(* IEC 61131-3 sources: AXOpen/src/showcase/app/src/core/AXOpen.AxoSequencer, 2 files *)

(* ---- AxoSequencerDocuExample.st ---- *)
USING AXOpen.Core;

NAMESPACE AxoSequencerExamples
    {S7.extern=ReadWrite}
    CLASS AxoSequencerDocuExample EXTENDS  AXOpen.Core.AxoObject
        VAR PUBLIC
            _mySequencer : AXOpen.Core.AxoSequencer;
            _step_1 : AxoStep;
            _step_2 : AxoStep;
            _step_3 : AxoStep;
            _myCounter : ULINT;
        END_VAR

        //<Initialize>
        METHOD PUBLIC Initialize
            _mySequencer.Run(THIS);
        END_METHOD
        //</Initialize>

        METHOD PUBLIC Execute
            //<Open>
            THIS.Initialize();
            IF _mySequencer.Open() THEN
                //All sequence logic needs to be placed inside the condition
                _myCounter := _myCounter + ULINT#1;

                IF _step_1.Execute(_mySequencer) THEN
                    IF (_myCounter > ULINT#50) THEN
                        _mySequencer.MoveNext();
                    END_IF;
                END_IF;

                IF _step_2.Execute(_mySequencer) THEN
                    IF (_myCounter > ULINT#100) THEN
                        _mySequencer.MoveNext();
                    END_IF;
                END_IF;

                IF _step_3.Execute(_mySequencer) THEN
                    IF (_myCounter > ULINT#150) THEN
                        _myCounter := ULINT#0;
                        _mySequencer.CompleteSequence();
                    END_IF;
                END_IF;
            END_IF;
            //</Open>
        END_METHOD

        METHOD StepExamples
            //<SimpleStep>
            IF _step_1.Execute(_mySequencer) THEN
                _myCounter := _myCounter + ULINT#1;
                // do something
                IF (_myCounter MOD ULINT#5) = ULINT#0 THEN
                    // continue to the next step of the sequence
                    _mySequencer.MoveNext();
                END_IF;
            END_IF;
            //</SimpleStep>

            //<EnableStep>
                IF _step_2.Execute(coord := _mySequencer, Enable := _myCounter <= ULINT#20) THEN
                    _myCounter := _myCounter + ULINT#1;
                    IF _myCounter = ULINT#20 THEN
                        // Jumping to step 1. As it is jumping backwards, the execution of step 1
                        // is going to be started in the next context cycle.
                        _mySequencer.RequestStep(_step_1);
                    END_IF;
                END_IF;
            //</EnableStep>

            //<FullStep>
                IF _step_3.Execute(coord := _mySequencer, Enable := TRUE, Description := '<#Process data#>' ) THEN
                    _myCounter := _myCounter + ULINT#1;
                    IF (_myCounter MOD ULINT#7) = ULINT#0 THEN
                        // Finalize the sequence and initiate the execution from the first step.
                        _mySequencer.CompleteSequence();
                    END_IF;
                END_IF;
            //</FullStep>
        END_METHOD

        //<SequenceMode>
        METHOD SequenceModeExamples
            // RunOnce: sequence executes once and stays in Done state
            _mySequencer.SequenceMode := eAxoSequenceMode#RunOnce;

            // Cyclic: sequence restarts automatically after CompleteSequence
            _mySequencer.SequenceMode := eAxoSequenceMode#Cyclic;
        END_METHOD
        //</SequenceMode>
    END_CLASS
END_NAMESPACE

(* ---- AxoSequencerExample.st ---- *)
USING AXOpen.Core;

NAMESPACE AxoSequencerExamples

    {S7.extern=ReadWrite}
    CLASS SequencerExample EXTENDS  AXOpen.Core.AxoObject
        VAR PUBLIC
            {#ix-set:AttributeName = "<#Sequencer example#>"}
            coord : AxoSequencer;
            Counter : ULINT;
            {#ix-set:AttributeName = "<#MicroStep-should be set to zero when entering new step#>"}
            MicroStep : UINT;
        END_VAR

        VAR PUBLIC
            {#ix-set:Description = "Step number one"}
            step_1 : AxoStep;
            {#ix-set:Description = "Step number two"}
            step_2 : AxoStep;
            {#ix-set:Description = "Step number three"}
            step_3 : AxoStep;
            {#ix-set:Description = "Step number four"}
            step_4 : AxoStep;
            {#ix-set:Description = "Step number five"}
            step_5 : AxoStep;
            {#ix-set:Description = "Step number six"}
            step_6 : AxoStep;
            {#ix-set:Description = "Step number seven"}
            step_7 : AxoStep;
            {#ix-set:Description = "Step number eight"}
            step_8 : AxoStep;
            {#ix-set:Description = "Step number nine"}
            step_9 : AxoStep;
            {#ix-set:Description = "Step number ten"}
            step_10 : AxoStep;
            Enable : ARRAY[1..10] OF BOOL :=[10(TRUE)];
        END_VAR

        METHOD PUBLIC Execute
            coord.Run(THIS);

            IF coord.Open() THEN

                IF(step_1.Execute(coord,Enable[1], 'Step_1')) THEN
                    IF step_1.IsFirstEntryToStep() THEN
                        Counter := ULINT#100;
                    END_IF;
                    Counter := Counter + ULINT#1;
                    IF(Counter >= ULINT#200 ) THEN
                        Counter := ULINT#0;
                        coord.MoveNext();
                    END_IF;
                END_IF;

                IF(step_2.Execute(coord,Enable[2], 'Step_2')) THEN
                    IF step_2.IsFirstEntryToStep() THEN
                        Counter := ULINT#200;
                    END_IF;
                    Counter := Counter + ULINT#1;
                    IF(Counter >= ULINT#300 ) THEN
                        Counter := ULINT#0;
                        coord.MoveNext();
                    END_IF;
                END_IF;

                IF(step_3.Execute(coord,Enable[3], 'Step_3')) THEN
                    IF step_3.IsFirstEntryToStep() THEN
                        Counter := ULINT#300;
                    END_IF;
                    Counter := Counter + ULINT#1;
                    IF(Counter >= ULINT#400 ) THEN
                        Counter := ULINT#0;
                        coord.MoveNext();
                    END_IF;
                END_IF;

                IF(step_4.Execute(coord,Enable[4], 'Step_4')) THEN
                    IF step_4.IsFirstEntryToStep() THEN
                        Counter := ULINT#400;
                    END_IF;
                    Counter := Counter + ULINT#1;
                    IF(Counter >= ULINT#500 ) THEN
                        Counter := ULINT#0;
                        coord.MoveNext();
                    END_IF;
                END_IF;

                IF(step_5.Execute(coord,Enable[5], 'Step_5')) THEN
                    IF step_5.IsFirstEntryToStep() THEN
                        Counter := ULINT#500;
                    END_IF;
                    Counter := Counter + ULINT#1;
                    IF(Counter >= ULINT#600 ) THEN
                        Counter := ULINT#0;
                        coord.MoveNext();
                    END_IF;
                END_IF;

                IF(step_6.Execute(coord,Enable[6], 'Step_6')) THEN
                    IF step_6.IsFirstEntryToStep() THEN
                        Counter := ULINT#600;
                    END_IF;
                    Counter := Counter + ULINT#1;
                    IF(Counter >= ULINT#700 ) THEN
                        Counter := ULINT#0;
                        coord.MoveNext();
                    END_IF;
                END_IF;

                IF(step_7.Execute(coord,Enable[7], 'Step_7')) THEN
                    IF step_7.IsFirstEntryToStep() THEN
                        Counter := ULINT#700;
                    END_IF;
                    Counter := Counter + ULINT#1;
                    IF(Counter >= ULINT#800 ) THEN
                        Counter := ULINT#0;
                        coord.RequestStep(step_1);
                        // coord.MoveNext();
                    END_IF;
                END_IF;

                IF(step_8.Execute(coord,Enable[8], 'Step_8')) THEN
                    IF step_8.IsFirstEntryToStep() THEN
                        Counter := ULINT#800;
                    END_IF;
                    Counter := Counter + ULINT#1;
                    IF(Counter >= ULINT#900 ) THEN
                        Counter := ULINT#0;
                        coord.MoveNext();
                    END_IF;
                END_IF;

                IF(step_9.Execute(coord,Enable[9], 'Step_9')) THEN
                    IF step_9.IsFirstEntryToStep() THEN
                        Counter := ULINT#900;
                    END_IF;
                    Counter := Counter + ULINT#1;
                    IF(Counter >= ULINT#1000 ) THEN
                        Counter := ULINT#0;
                        coord.MoveNext();
                    END_IF;
                END_IF;

                IF(step_10.Execute(coord,Enable[10], 'Step_10')) THEN
                    IF step_10.IsFirstEntryToStep() THEN
                        Counter := ULINT#1000;
                    END_IF;
                    Counter := Counter + ULINT#1;
                    IF(Counter >= ULINT#1100 ) THEN
                        Counter := ULINT#0;
                        coord.CompleteSequence();
                    END_IF;
                END_IF;
                coord.SetMicroStepValue(coord.GetMicroStepValue() + UINT#2);
                MicroStep := coord.GetMicroStepValue();
            END_IF;

        END_METHOD
    END_CLASS
END_NAMESPACE
